(* IEC 61131-3 sources: ATCMcontrol_Engineering/src/Target/ATHW119/Libs/ATCM_IEC1131_3/table_37, 3 files *)

(* ---- tof.st ---- *)
(*[[
    UserURL= "ATCMfile:TOF.htm"
]]*)

FUNCTION_BLOCK TOF

VAR_INPUT   (* Inputs *)
    IN : BOOL := FALSE; (* Input        *)
    PT : TIME := T#0s;  (* Preset time  *)
END_VAR

VAR_OUTPUT  (* Outputs *)
    Q  : BOOL := FALSE; (* FALSE if ET >= PT *)
    ET : TIME := T#0s; (* Elapsed time      *)
END_VAR

VAR NON_RETAIN
    StartTime : TIME;
    State : INT := 0;
END_VAR

VAR
    M         : BOOL := FALSE;
END_VAR

inline { STDLIB(tof) }

END_FUNCTION_BLOCK

(* ---- ton.st ---- *)
(*[[
   UserURL= "ATCMfile:TON.htm"
]]*)

FUNCTION_BLOCK TON

VAR_INPUT   (* Inputs *)
    IN : BOOL := FALSE; (* Input        *)
    PT : TIME := T#0s;  (* Preset time 	*)
END_VAR

VAR_OUTPUT  (* Outputs *)
    Q  : BOOL := FALSE; (* TRUE if ET >= PT *)
    ET : TIME := T#0s;  (* Elapsed time     *)
END_VAR

VAR NON_RETAIN
    StartTime : TIME;
    State : INT := 0;
END_VAR

VAR
    M         : BOOL := FALSE;
END_VAR

inline { STDLIB(ton) }

END_FUNCTION_BLOCK

(* ---- tp.st ---- *)
(*[[
    UserURL= "ATCMfile:TP.htm"
]]*)

FUNCTION_BLOCK TP

VAR_INPUT   (* Inputs *)
    IN : BOOL := FALSE; (* Input       *)
    PT : TIME := T#0s;  (* Preset time *)
END_VAR

VAR_OUTPUT  (* Outputs *)
    Q  : BOOL := FALSE; (* FALSE if ET >= PT    *)
    ET : TIME := T#0s;  (* Elapsed time         *)
END_VAR

VAR NON_RETAIN
    StartTime : TIME;
    State     : INT := 0;
END_VAR

VAR
    M         : BOOL := FALSE;
END_VAR

inline { STDLIB(tp) }

END_FUNCTION_BLOCK
